{attribute 'no_explicit_call' := 'do not call this function block directly'} 
{attribute 'enable_dynamic_creation'}
FUNCTION_BLOCK PointerDictionaryEnumerator EXTENDS PointerBasedEnumerator
VAR
	_ClassName : STRING := __POUNAME();
	_Dictionary : IReadOnlyPointerDictionary;
	_Current : KEY_VALUE_POINTER_PAIR;
END_VAR

{attribute 'monitoring' := 'call'}
PROPERTY ClassName : STRING
GET
ClassName := _ClassName;
END_GET
END_PROPERTY

{attribute 'OPC.UA.DA.Property' := '1'}
{attribute 'monitoring' := 'call'}
PROPERTY Current : PVOID
GET
Current := ADR(_Current);
END_GET
END_PROPERTY

{attribute 'OPC.UA.DA.Property' := '1'}
{attribute 'monitoring' := 'call'}
PROPERTY CurrentKeyValuePair : POINTER TO KEY_VALUE_POINTER_PAIR
GET
CurrentKeyValuePair := ADR(_Current);
END_GET
END_PROPERTY

METHOD INTERNAL Initialize 
VAR_INPUT
	dictionary : IReadOnlyPointerDictionary;
END_VAR
_Dictionary := dictionary;
END_METHOD

{attribute "object_name" := "MoveNext"}
METHOD MoveNext : BOOL
_CurrentIndex := _CurrentIndex + 1;

IF _CurrentIndex >= _Dictionary.Count THEN
	_Current.Key := 0;
	_Current.Value := 0;

	_CurrentIndex := _Dictionary.Count;
ELSE
	_Current.Key := _Dictionary.GetKeyByIndex(_CurrentIndex);
	_Current.Value := _Dictionary.GetValueByIndex(_CurrentIndex);
	
	MoveNext := TRUE;
END_IF
END_METHOD

{attribute "object_name" := "Reset"}
METHOD Reset
SUPER^.Reset();

_Current.Key := 0;
_Current.Value := 0;
END_METHOD

{attribute 'monitoring' := 'call'}
PROPERTY Size : ULINT
GET
Size := XSIZEOF(THIS^);
END_GET
END_PROPERTY

END_FUNCTION_BLOCK

(* stored: Version 1.1.0.1
   POU PointerDictionaryEnumerator: Id {0f27f47a-acdb-023c-212e-33c787813e08}, SpecialFunc None
   Property ClassName: Id {dc1ed2eb-dc27-09f1-0152-a7c860443582}
   Get Get: Id {7e542f89-2072-0a03-2838-c1ebbaaea807}
   Property Current: Id {a559bb7d-ff89-0905-2cce-1f77e5a90617}
   Get Get: Id {1192bef5-1645-075c-0a47-f6ed4ad79ada}
   Property CurrentKeyValuePair: Id {16b41111-8c37-07df-2111-1c67d5814b7f}
   Get Get: Id {e59bd0cb-d42d-04d7-0e91-e5935a47d47f}
   Method Initialize: Id {b838ba5e-1e12-017d-0ba1-23a086e939c4}
   Method MoveNext: Id {87be4302-a7c3-0049-1efc-84335818745a}
   Method Reset: Id {ca9926ff-ba9d-08fd-2694-f9c502a79fbc}
   Property Size: Id {26880d90-bdfb-4ffe-a7d1-e0f62465df06}
   Get Get: Id {1908b89d-f98b-4de3-a04a-40488af16791} *)
